Fanuc KAREL source: kt00911.KL

-- PROVISIONAL review KL for V940-1; original PC SHA256 8606246cf7e4ba7e33e3e2f96ddc3895715fab99c4eee3371bb84f807a90f73c
-- Incomplete behavior may be omitted. Consult companion uncertainty JSON. Do not deploy.
PROGRAM KT00911
%NOLOCKGROUP
BEGIN
  -- V9_ZERO_TABLE_METADATA_HINT layout=0002_ascii; no indexed target words; source/name/runtime held
  -- UNRESOLVED_PC offsets 5-31; opcodes 27,27,49,7E,AD,31,4A
  -- UNRESOLVED_PC offsets 36-40; opcodes 7F
END KT00911
